FUNCTION_BLOCK FB_Valve
VAR_INPUT
	command : BOOL ;
	feedback : BOOL ;
	auto_man : BOOL ;
	time_feedback : INT ;
END_VAR
VAR_OUTPUT
	valve: BOOL;	
END_VAR
VAR
	fbTimer: TON;
	fail : BOOL ;
END_VAR

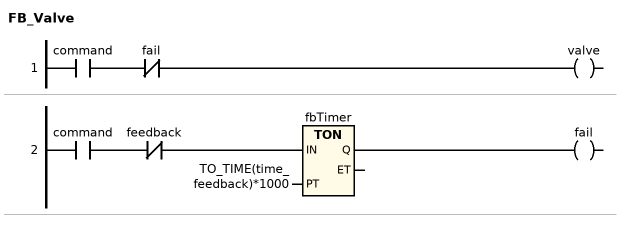
// NETWORK 1
valve := command AND NOT fail;

// NETWORK 2
fbTimer(IN := command AND NOT feedback, PT := TO_TIME(time_feedback)*1000); // TON
fail := fbTimer.Q;

END_FUNCTION_BLOCK

(* stored: Version 1.1.0.1, ProductVersion 3.1.4024.12
   POU FB_Valve: Id {14010fce-d78d-40fc-abcc-ef8375c3b976}, SpecialFunc None *)
